Staubli VAL3: action_resume.pgx

program action_resume()
begin
  //
  // suspend all the task action
  //
  // check first...
  if taskStatus("Cycle")!=-1
    taskResume("Cycle",0)
  endIf
  if taskStatus("Action")!=-1
    taskResume("Action",0)
  endIf
  //..
end
